// TIA Portal V18 export
VAR_GLOBAL   // PLC tag table "Input"
   "Driver Alarm Left input" AT %I0.0 : Bool;
   "Driver Fault Left input" AT %I0.1 : Bool;
   "Driver Alarm Right input" AT %I0.2 : Bool;
   "Driver Fault Right input" AT %I0.3 : Bool;
   "Cab Driver Alarm input" AT %I0.4 : Bool;
   "Cab Driver Fault input" AT %I0.5 : Bool;
   "Rotunda Fire Detector input" AT %I0.6 : Bool;
   "GPU1 Active input" AT %I0.7 : Bool;
   "Drive Wheel Fuse input" AT %I2.0 : Bool;
   "Fuse Hydraulic input" AT %I2.3 : Bool;
   "Cab Fuse input" AT %I2.4 : Bool;
   "Phase Relay input" AT %I2.5 : Bool;
   "Rotunda LSW Left Stop input" AT %I3.0 : Bool;
   "Rotunda LSW Right Stop input" AT %I3.1 : Bool;
   "Tunnel LSW FW Slow İnput" AT %I3.2 : Bool;   // FW Slow
   "Tunnel LSW BW Slow İnput" AT %I3.3 : Bool;   // BW Slow
   "Tunnel LSW FW Stop İnput" AT %I3.4 : Bool;   // FW Stop
   "Tunnel LSW BW Stop İnput" AT %I3.5 : Bool;   // BW Stop
   "Tunnel LSW FW Em Stop İnput" AT %I3.6 : Bool;   // FW Em Stop
   "Tunnel LSW BW Em Stop İnput" AT %I3.7 : Bool;   // BW Em Stop
   "Drive LSW Stop Left input" AT %I4.0 : Bool;
   "Drive LSW Stop Right input" AT %I4.1 : Bool;
   "SafetyEdge Relay input" AT %I4.2 : Bool;   // Box in Relay Reset
   "SafetyEdge Aux input" AT %I4.3 : Bool;   // Edge touch
   "Em Stop Left input" AT %I4.4 : Bool;
   "Em Stop Right input" AT %I4.5 : Bool;
   "Cabin LSW Left input" AT %I5.2 : Bool;
   "Cabin LSW Right input" AT %I5.3 : Bool;
   "UltraSonic for AirCraft input" AT %I5.4 : Bool;
   "UltraSonic for Object input" AT %I5.5 : Bool;
   "PhotoCell for AirCraft input" AT %I5.6 : Bool;
   "Bumper Touch Left input" AT %I5.7 : Bool;
   "Bumper Touch Mid input" AT %I6.0 : Bool;
   "Bumper Touch Right input" AT %I6.1 : Bool;
   "Canopy Touch Left input" AT %I6.2 : Bool;
   "Canopy Touch Right input" AT %I6.3 : Bool;
   "AutoLeveller Up Sensor input" AT %I6.7 : Bool;
   "AutoLeveller Down Sensor input" AT %I7.0 : Bool;
   "Fuse 2Power Supply input" AT %I8.0 : Bool;
   "PCA Active input" AT %I8.1 : Bool;
   "Fuse 1Power Supply input" AT %I8.2 : Bool;
   "AutoLeveller Touch input" AT %I8.3 : Bool;
   "GPU2 Active input" AT %I8.4 : Bool;
   "Fire Detector Cabin input" AT %I8.5 : Bool;
   "Fuse Hose Ritriver input" AT %I8.6 : Bool;
   "Fuse MC input" AT %I8.7 : Bool;
   "Hose Active input" AT %I9.0 : Bool;
   "GPU1 Error input" AT %I9.1 : Bool;
   "PCA Error input" AT %I9.2 : Bool;
   "GPU2 Error input" AT %I9.3 : Bool;
   "SafetyShoe Relay input" AT %I10.0 : Bool;
   "SafetyShoe Aux input" AT %I10.1 : Bool;
   "Fuse AutoLeveller input" AT %I10.2 : Bool;
   "Fuse Left Canopy input" AT %I10.4 : Bool;
   "Fuse Right Canopy input" AT %I10.5 : Bool;
   "Fuse Cab Floor input" AT %I10.6 : Bool;
   "Button ByPass input" AT %I11.0 : Bool;
   "Button Reset input" AT %I11.1 : Bool;
   "Button Light Int input" AT %I11.2 : Bool;
   "Button Ext Light input" AT %I11.3 : Bool;
   "Button Ext Projector input" AT %I11.4 : Bool;
   "Em Stop Button input" AT %I11.5 : Bool;
   "Key-1 ON input" AT %I11.6 : Bool;
   "Key-2 OFF input" AT %I11.7 : Bool;
   "Cab Button Left input" AT %I12.0 : Bool;
   "Cab Button Right input" AT %I12.1 : Bool;
   "Button PBB Up input" AT %I12.2 : Bool;
   "Button Pbb Down input" AT %I12.3 : Bool;
   "Canopy Button FW input" AT %I12.5 : Bool;
   "Canopy Button BW input" AT %I12.4 : Bool;
   "Cab Floor FW input" AT %I12.6 : Bool;
   "Cab Floor BW input" AT %I12.7 : Bool;
   "JoyStick X33 FW input" AT %I13.3 : Bool;
   "JoyStick X22 L2 input" AT %I13.4 : Bool;
   "JoyStick X44 L3 input" AT %I13.5 : Bool;
   "JoyStick X55 BW input" AT %I13.6 : Bool;
   "JoyStick Y33 RGHT input" AT %I13.7 : Bool;
   "JoyStick Y22 L2 input" AT %I14.0 : Bool;
   "JoyStick Y44 L3 input" AT %I14.1 : Bool;
   "JoyStick Y55 LFT input" AT %I14.2 : Bool;
   "JoyStick 91 Brake input" AT %I14.3 : Bool;
   "SafetyShoe Box Status input" AT %I6.4 : Bool;
END_VAR
